// TIA Portal V17 export
// export: Created 2023-02-14T02:49:45.987409Z, ExportSetting WithDefaults, DisplayName Totally Integrated Automation Portal, DisplayVersion V17, DisplayName TIA Portal Openness, DisplayVersion V17, DisplayName TIA Portal Teamcenter Gateway, DisplayVersion V17, DisplayName TIA Portal Version Control Interface, DisplayVersion V17, DisplayName SINAMICS Startdrive Advanced, DisplayVersion V17, DisplayName SINAMICS Startdrive G130, G150, S120, S150, SINAMICS MV, S210, DisplayVersion V17, DisplayName SINAMICS Startdrive G110M, G120, G120C, G120D, G120P, G115D, DisplayVersion V17, DisplayName STEP 7 Professional, DisplayVersion V17, DisplayName STEP 7 Safety, DisplayVersion V17, DisplayName WinCC Professional, DisplayVersion V17
DATA_BLOCK "Sim_PTS_DB"   // DB1001
VERSION : 0.1
// stored: AutoNumber false, DBAccessibleFromOPCUA true, DBAccessibleFromWebserver true, InstanceOfName Sim_PT1, InstanceOfType FB
"Sim_PT1"
   // VAR_INPUT
   //    Reset : Bool;
   //    Calc_Param : Bool;
   //    Input : Real;
   //    TM_LAG1 : Real;
   //    GAIN : Real;
   //    Cycle : Real;
   //    Max_Out : Real;
   //    AMB_TEM : Real;
   // END_VAR
   // VAR_OUTPUT
   //    Max_reached : Bool;
   //    Output : Real;
   // END_VAR
   // VAR
   //    r_f1 : Real;
   //    r_e1 : Real;
   //    overfirst : Bool;
   // END_VAR
BEGIN
END_DATA_BLOCK
